Omron Sysmac Studio project TicTacToe8winnerrowline (Sysmac Studio 1.56.0.64011, StandardProject)

# Controller new_Controller_0: NJ501-1500 version 1.64
Units and slaves: Power Supply : NJ-Px3001; CPU : NJ501-1500
Task PrimaryTask (priority 4, period or condition 1000): Program0

VAR_GLOBAL
    Restart : BOOL := False;
    Winner : INT := 0;
    CurrentPlayer : INT := 1;
    Board : ARRAY[0..8] OF INT := [0,0,0,0,0,0,0,0,0];
    Button_1 : BOOL := False;
    Button_2 : BOOL := False;
    Button_3 : BOOL := False;
    Button_4 : BOOL := False;
    Button_5 : BOOL := False;
    Button_6 : BOOL := False;
    Button_7 : BOOL := False;
    Button_8 : BOOL := False;
    Button_9 : BOOL := False;
    WinnerMessage : DINT := 0;
    GameStatus : STRING[255] := '';
    Button_0 : BOOL := False;
    ButtonText : ARRAY[0..8] OF STRING[2];
    ButtonText0 : STRING[255] := '';
    ButtonText1 : STRING[255] := '';
    ButtonText2 : STRING[255] := '';
    ButtonText3 : STRING[255] := '';
    ButtonText4 : STRING[255] := '';
    ButtonText5 : STRING[255] := '';
    ButtonText6 : STRING[255] := '';
    ButtonText7 : STRING[255] := '';
    ButtonText8 : STRING[255] := '';
    LineRow1 : BOOL := False;
    LineRow2 : BOOL := False;
    LineRow3 : BOOL := False;
    LineCol1 : BOOL := False;
    LineCol2 : BOOL := False;
    LineCol3 : BOOL := False;
    LineDiag2 : BOOL := False;
    LineDiag1 : BOOL := False;
END_VAR

PROGRAM Program0
VAR
    i : INT;
    j : INT;
END_VAR
VAR_EXTERNAL
    Restart : BOOL;
    Winner : INT;
    CurrentPlayer : INT;
    Board : ARRAY[0..8] OF INT;
    Button_1 : BOOL;
    Button_2 : BOOL;
    Button_3 : BOOL;
    Button_4 : BOOL;
    Button_5 : BOOL;
    Button_6 : BOOL;
    Button_7 : BOOL;
    Button_8 : BOOL;
    Button_9 : BOOL;
    WinnerMessage : DINT;
    GameStatus : STRING[255];
    ButtonText : ARRAY[0..8] OF STRING[2];
    ButtonText0 : STRING[255];
    ButtonText1 : STRING[255];
    ButtonText2 : STRING[255];
    ButtonText3 : STRING[255];
    ButtonText4 : STRING[255];
    ButtonText5 : STRING[255];
    ButtonText6 : STRING[255];
    ButtonText7 : STRING[255];
    ButtonText8 : STRING[255];
    LineRow1 : BOOL;
    LineRow2 : BOOL;
    LineRow3 : BOOL;
    LineCol1 : BOOL;
    LineCol2 : BOOL;
    LineCol3 : BOOL;
    LineDiag1 : BOOL;
    LineDiag2 : BOOL;
END_VAR

(* Section Section0: ladder, written here as Structured Text *)

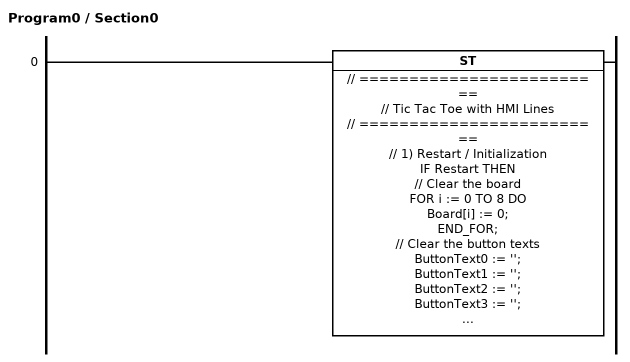
(* Rung 0 *)
// =========================
// Tic Tac Toe with HMI Lines
// =========================

// 1) Restart / Initialization
IF Restart THEN
    // Clear the board
    FOR i := 0 TO 8 DO
        Board[i] := 0;
    END_FOR;

    // Clear the button texts
    ButtonText0 := '';
    ButtonText1 := '';
    ButtonText2 := '';
    ButtonText3 := '';
    ButtonText4 := '';
    ButtonText5 := '';
    ButtonText6 := '';
    ButtonText7 := '';
    ButtonText8 := '';

    // Reset game status variables
    Winner := 0;
    WinnerMessage := 0;
    GameStatus := '';
    CurrentPlayer := 1;

    // Reset line indicators
    LineRow1 := FALSE;
    LineRow2 := FALSE;
    LineRow3 := FALSE;
    LineCol1 := FALSE;
    LineCol2 := FALSE;
    LineCol3 := FALSE;
    LineDiag1 := FALSE;
    LineDiag2 := FALSE;

    // Turn off Restart to avoid re-trigger
    Restart := FALSE;
END_IF;


// 2) Allow moves only if no winner yet
IF Winner = 0 THEN
    // Player Move Handling
    IF Button_1 AND (Board[0] = 0) THEN
        Board[0] := CurrentPlayer;
        IF CurrentPlayer = 1 THEN
            ButtonText0 := 'X';
        ELSE
            ButtonText0 := 'O';
        END_IF;
        CurrentPlayer := 3 - CurrentPlayer;
    END_IF;

    IF Button_2 AND (Board[1] = 0) THEN
        Board[1] := CurrentPlayer;
        IF CurrentPlayer = 1 THEN
            ButtonText1 := 'X';
        ELSE
            ButtonText1 := 'O';
        END_IF;
        CurrentPlayer := 3 - CurrentPlayer;
    END_IF;

    IF Button_3 AND (Board[2] = 0) THEN
        Board[2] := CurrentPlayer;
        IF CurrentPlayer = 1 THEN
            ButtonText2 := 'X';
        ELSE
            ButtonText2 := 'O';
        END_IF;
        CurrentPlayer := 3 - CurrentPlayer;
    END_IF;

    IF Button_4 AND (Board[3] = 0) THEN
        Board[3] := CurrentPlayer;
        IF CurrentPlayer = 1 THEN
            ButtonText3 := 'X';
        ELSE
            ButtonText3 := 'O';
        END_IF;
        CurrentPlayer := 3 - CurrentPlayer;
    END_IF;

    IF Button_5 AND (Board[4] = 0) THEN
        Board[4] := CurrentPlayer;
        IF CurrentPlayer = 1 THEN
            ButtonText4 := 'X';
        ELSE
            ButtonText4 := 'O';
        END_IF;
        CurrentPlayer := 3 - CurrentPlayer;
    END_IF;

    IF Button_6 AND (Board[5] = 0) THEN
        Board[5] := CurrentPlayer;
        IF CurrentPlayer = 1 THEN
            ButtonText5 := 'X';
        ELSE
            ButtonText5 := 'O';
        END_IF;
        CurrentPlayer := 3 - CurrentPlayer;
    END_IF;

    IF Button_7 AND (Board[6] = 0) THEN
        Board[6] := CurrentPlayer;
        IF CurrentPlayer = 1 THEN
            ButtonText6 := 'X';
        ELSE
            ButtonText6 := 'O';
        END_IF;
        CurrentPlayer := 3 - CurrentPlayer;
    END_IF;

    IF Button_8 AND (Board[7] = 0) THEN
        Board[7] := CurrentPlayer;
        IF CurrentPlayer = 1 THEN
            ButtonText7 := 'X';
        ELSE
            ButtonText7 := 'O';
        END_IF;
        CurrentPlayer := 3 - CurrentPlayer;
    END_IF;

    IF Button_9 AND (Board[8] = 0) THEN
        Board[8] := CurrentPlayer;
        IF CurrentPlayer = 1 THEN
            ButtonText8 := 'X';
        ELSE
            ButtonText8 := 'O';
        END_IF;
        CurrentPlayer := 3 - CurrentPlayer;
    END_IF;
END_IF;


// 3) Win Detection Logic
// Check rows
IF (Board[0] = Board[1]) AND (Board[1] = Board[2]) AND (Board[0] <> 0) THEN
    Winner := Board[0];
    LineRow1 := TRUE; // Activate line for top row
END_IF;
IF (Board[3] = Board[4]) AND (Board[4] = Board[5]) AND (Board[3] <> 0) THEN
    Winner := Board[3];
    LineRow2 := TRUE; // Middle row
END_IF;
IF (Board[6] = Board[7]) AND (Board[7] = Board[8]) AND (Board[6] <> 0) THEN
    Winner := Board[6];
    LineRow3 := TRUE; // Bottom row
END_IF;

// Check columns
IF (Board[0] = Board[3]) AND (Board[3] = Board[6]) AND (Board[0] <> 0) THEN
    Winner := Board[0];
    LineCol1 := TRUE; // Left column
END_IF;
IF (Board[1] = Board[4]) AND (Board[4] = Board[7]) AND (Board[1] <> 0) THEN
    Winner := Board[1];
    LineCol2 := TRUE; // Middle column
END_IF;
IF (Board[2] = Board[5]) AND (Board[5] = Board[8]) AND (Board[2] <> 0) THEN
    Winner := Board[2];
    LineCol3 := TRUE; // Right column
END_IF;

// Check diagonals
IF (Board[0] = Board[4]) AND (Board[4] = Board[8]) AND (Board[0] <> 0) THEN
    Winner := Board[0];
    LineDiag1 := TRUE; // Main diagonal
END_IF;
IF (Board[2] = Board[4]) AND (Board[4] = Board[6]) AND (Board[2] <> 0) THEN
    Winner := Board[2];
    LineDiag2 := TRUE; // Other diagonal
END_IF;


// 4) Update WinnerMessage & GameStatus
IF Winner = 1 THEN
    WinnerMessage := 1; // Player 1 Wins
    GameStatus := 'Player 1 Wins!';

ELSIF Winner = 2 THEN
    WinnerMessage := 2; // Player 2 Wins
    GameStatus := 'Player 2 Wins!';

ELSIF (Board[0] <> 0 AND Board[1] <> 0 AND Board[2] <> 0 AND
       Board[3] <> 0 AND Board[4] <> 0 AND Board[5] <> 0 AND
       Board[6] <> 0 AND Board[7] <> 0 AND Board[8] <> 0 AND (Winner = 0)) THEN
    WinnerMessage := 0; // It's a Draw
    GameStatus := 'It is a Draw!';
END_IF;
END_PROGRAM

# Device HMI_NA5_0 (NA): not converted